(* IEC 61131-3 sources: netflux/Codesys_V3/NETFLUX, 14 files *)

(* ---- DUT_INPUTS.st ---- *)
TYPE DUT_INPUTS :
STRUCT
	Conv1_fb_pulse : BIT; //Pulse position sensor
	conv2_fb_pulse : BIT; //Pulse position sensor
	SPARE_INPUT_01 : BIT; //Spare bit
	SPARE_INPUT_02 : BIT; //Spare bit
	SPARE_INPUT_03 : BIT; //Spare bit
	SPARE_INPUT_04 : BIT; //Spare bit
	SPARE_INPUT_05 : BIT; //Spare bit
	SPARE_INPUT_06 : BIT; //Spare bit
	PS1_fb : BIT; //Sensor feedback signal
	PS2_fb : BIT; //Sensor feedback signal
	SPARE_INPUT_07 : BIT; //Spare bit
	SPARE_INPUT_08 : BIT; //Spare bit
	SPARE_INPUT_09 : BIT; //Spare bit
	SPARE_INPUT_10 : BIT; //Spare bit
	SPARE_INPUT_11 : BIT; //Spare bit
	SPARE_INPUT_12 : BIT; //Spare bit
	RDS1_fb_rised : BIT; //Rising divert at raised position
	RDS1_fb_initial : BIT; //Rising divert at initial position
	SPARE_INPUT_13 : BIT; //Spare bit
	SPARE_INPUT_14 : BIT; //Spare bit
	SPARE_INPUT_15 : BIT; //Spare bit
	SPARE_INPUT_16 : BIT; //Spare bit
	SPARE_INPUT_17 : BIT; //Spare bit
	SPARE_INPUT_18 : BIT; //Spare bit
	SPARE_INPUT_19 : BIT; //Spare bit
	SPARE_INPUT_20 : BIT; //Spare bit
	SPARE_INPUT_21 : BIT; //Spare bit
	SPARE_INPUT_22 : BIT; //Spare bit
	SPARE_INPUT_23 : BIT; //Spare bit
	SPARE_INPUT_24 : BIT; //Spare bit
	SPARE_INPUT_25 : BIT; //Spare bit
	SPARE_INPUT_26 : BIT; //Spare bit
	SPARE_INPUT_27 : BIT; //Spare bit
	SPARE_INPUT_28 : BIT; //Spare bit
	SPARE_INPUT_29 : BIT; //Spare bit
	SPARE_INPUT_30 : BIT; //Spare bit

END_STRUCT
END_TYPE

(* ---- DUT_OUTPUTS.st ---- *)
TYPE DUT_OUTPUTS :
STRUCT
	Conv1_cmd_fwd : BIT; //Run conveyor forward
	conv2_cmd_fwd : BIT; //Run conveyor forward
	Conv1_cmd_bwd : BIT; //Run conveyor backward
	conv2_cmd_bwd : BIT; //Run conveyor backward
	SPARE_OUTPUT_01 : BIT; //Spare bit
	SPARE_OUTPUT_02 : BIT; //Spare bit
	SPARE_OUTPUT_03 : BIT; //Spare bit
	SPARE_OUTPUT_04 : BIT; //Spare bit
	em1_cmd_emit : BIT; //Trigger item spawn
	destroyer_cmd_on : BIT; //Enable destroyer
	SPARE_OUTPUT_05 : BIT; //Spare bit
	SPARE_OUTPUT_06 : BIT; //Spare bit
	SPARE_OUTPUT_07 : BIT; //Spare bit
	SPARE_OUTPUT_08 : BIT; //Spare bit
	SPARE_OUTPUT_09 : BIT; //Spare bit
	SPARE_OUTPUT_10 : BIT; //Spare bit
	RDS1_cmd_left : BIT; //Command divert left (belt forward)
	RDS1_cmd_right : BIT; //Command divert right (belt backward)
	SPARE_OUTPUT_11 : BIT; //Spare bit
	SPARE_OUTPUT_12 : BIT; //Spare bit
	SPARE_OUTPUT_13 : BIT; //Spare bit
	SPARE_OUTPUT_14 : BIT; //Spare bit
	SPARE_OUTPUT_15 : BIT; //Spare bit
	SPARE_OUTPUT_16 : BIT; //Spare bit
	SPARE_OUTPUT_17 : BIT; //Spare bit
	SPARE_OUTPUT_18 : BIT; //Spare bit
	SPARE_OUTPUT_19 : BIT; //Spare bit
	SPARE_OUTPUT_20 : BIT; //Spare bit
	SPARE_OUTPUT_21 : BIT; //Spare bit
	SPARE_OUTPUT_22 : BIT; //Spare bit
	SPARE_OUTPUT_23 : BIT; //Spare bit
	SPARE_OUTPUT_24 : BIT; //Spare bit
	SPARE_OUTPUT_25 : BIT; //Spare bit
	SPARE_OUTPUT_26 : BIT; //Spare bit

END_STRUCT
END_TYPE

(* ---- DUT_RECV_DATA.st ---- *)
{attribute 'pack_mode' := '0'}
TYPE DUT_RECV_DATA :
STRUCT
		byteArray :	ARRAY[0..50] OF BYTE;
		some_INT :	INT;
		some_TIME :	TIME;
		some_REAL :	REAL;
		b1 :	BYTE ;
		b2 :	BYTE ;
		b3 :	BYTE ;

END_STRUCT
END_TYPE

(* ---- ENUM_NetfluxSocketState.st ---- *)
TYPE ENUM_NetfluxSocketState :
(
    IDLE := 0,
    CREATE := 10,
    BIND := 20,
    NONBLOCK := 30,
    RUNNING := 40,
    ERROR := 99
) INT;
END_TYPE

(* ---- GVL.st ---- *)
{attribute 'qualified_only'}
VAR_GLOBAL
	data_send :  DUT_OUTPUTS;
	data_recv :  DUT_INPUTS;
END_VAR

(* ---- fbNetflux_Recieve.st ---- *)
(*
    Function Block: fbPUDP_Recieve
    Description: Manages the receiving part of a UDP communication.
                 It uses a sequence number to discard duplicate or out-of-order packets
                 and a watchdog timer to detect communication loss. It provides outputs
                 needed by a corresponding Send block.
*)
FUNCTION_BLOCK fbNetflux_Recieve
VAR_INPUT
    // --- Connection Parameters ---
    i_uiLocalPort : UINT;   // Local UDP port to listen on.

    // --- Data Reception Parameters ---
	i_ptrReceiveData : POINTER TO BYTE; // Pointer to the destination buffer where the received data payload will be stored.
	i_uiSizeReceiveData : UINT;         // The exact size of the data payload to copy. The user is responsible for ensuring this size matches the sender's payload.

    // --- Watchdog Parameters ---
    i_tWatchInterval : TIME := T#1S;    // Watchdog timeout. If no new valid packet arrives within this interval, o_bError is set.
    i_xKeepValuesOnTimeout : BOOL;      // If TRUE, the last received values are kept in the destination buffer on watchdog timeout. If FALSE, the buffer is cleared for safety.
END_VAR
VAR_OUTPUT
    o_xError: BOOL;        // Becomes TRUE if no valid packet has been received, if the watchdog has timed out, or if a library error occurs.
    o_eErrorID: NBS.ERROR; // Propagates the specific error code from the underlying NBS library if an error occurs.
	o_hPeer: LWORD;         // Outputs the handle of the UDP peer. This is required by the corresponding Send block to use the same socket.
	o_bPartnerSeqNumber : BYTE; // Outputs the last received sequence number from the partner. This is needed by the Send block to send it back as a feedback sequence number.
	o_bCurrentFeedbackSeqNumber : BYTE; // Stores the feedback sequence number from the current valid packet. Used by the watchdog.
END_VAR
VAR
	// --- Internal state flags ---
	s_xFirstPacketReceived : BOOL;      // Flag to track if at least one valid packet has been received since startup or last timeout.
    s_xWatchdogTimeout : BOOL;          // Flag set by the watchdog timer when no new packet arrives in time.

    // --- UDP library instances ---
    s_fbPeer: NBS.UDP_Peer := (xEnable := TRUE); // Manages the UDP socket itself.
	s_fbUDPReceive : NBS.UDP_Receive;            // Handles the continuous reception of data into the internal buffer.
    s_tonWatchdog : TON;                         // Watchdog timer to detect communication loss.

    // --- Internal receive buffer ---
    s_aRecvBuffer: ARRAY[0..1460] OF BYTE;       // Raw buffer that receives the entire UDP packet.
	s_ptrRecvBuffer : POINTER TO BYTE := ADR(s_aRecvBuffer);
	s_szRecvBuffer : UINT := SIZEOF(s_aRecvBuffer);

	// --- Sequence number handling ---
	s_bPreviousRecvSeqNumber : BYTE;    // Stores the sequence number of the last processed packet to detect new ones.

    s_bPreviousFeedbackSeqNumber : BYTE;// Stores the feedback sequence number from the previous cycle to detect changes.
END_VAR
VAR_TEMP
    xIsNewPacket : BOOL;                // Temporary flag to indicate if a received packet is newer than the last processed one.
END_VAR

// === IMPLEMENTATION ===
(*
    This function block receives data via UDP and writes it into a specified destination buffer.

    Expected UDP Payload Structure:
    - Byte 0: Sequence Number (rolls over from 255 to 0). Used to identify new/unique packets.
    - Byte 1: Feedback Sequence Number. A copy of the sender's own receive sequence number. Used here for the watchdog.
    - Byte 2...N: The actual data payload.

    How it works:
    1. It continuously listens for incoming UDP packets on the specified port using the NBS library blocks.
    2. It checks for a new packet by comparing the sequence number (Byte 0) of the incoming packet with the last one processed.
    3. A robust sequence number validation handles counter wrap-around and rejects old, duplicate, or out-of-order packets.
    4. For valid new packets, a fixed-size data payload (defined by 'i_uiSizeReceiveData') is copied from the internal buffer to the user-provided destination buffer.
    5. A watchdog timer monitors the reception of valid packets. If no new packet arrives within 'i_tWatchInterval', an error is flagged.
    6. If the watchdog expires, the behavior is controlled by 'i_bKeepValuesOnTimeout' (either clear the destination buffer or keep the last valid data).
*)

// 1. Initialize and open the UDP Peer on the specified local port.
s_fbPeer(uiPort:=i_uiLocalPort);
// 1a. Output the peer handle so a corresponding Send block can use the same socket.
o_hPeer := s_fbPeer.hPeer;

// 2. Execute the UDP_Receive instruction to listen for data. This block continuously updates s_aRecvBuffer with the latest received packet.
s_fbUDPReceive(
	xEnable:= s_fbPeer.xActive,
	hPeer:= s_fbPeer.hPeer,
	szSize:= s_szRecvBuffer,
	pData:= s_ptrRecvBuffer);

// 3. Check for a new packet by detecting a change in the sequence number byte.
IF s_aRecvBuffer[0] <> s_bPreviousRecvSeqNumber THEN
	// 3a. Pass the received sequence number to the output immediately. The Send block will use this for feedback.
	o_bPartnerSeqNumber := s_aRecvBuffer[0];

    // A packet with a different sequence number has arrived.
    // Now, validate if it's logically NEWER than the last one, handling the 8-bit counter wrap-around.
    // This prevents processing old packets that may arrive out of order.
    // A packet is considered "new" if it's the first one, its number is slightly ahead, or it has wrapped around.
    xIsNewPacket := NOT s_xFirstPacketReceived OR
        (s_aRecvBuffer[0] > s_bPreviousRecvSeqNumber AND s_aRecvBuffer[0] - s_bPreviousRecvSeqNumber < 128) OR
        (s_aRecvBuffer[0] < s_bPreviousRecvSeqNumber AND s_bPreviousRecvSeqNumber - s_bPreviousRecvSeqNumber > 128);

	IF xIsNewPacket THEN
        // --- Process Valid New Packet ---
        s_xFirstPacketReceived := TRUE;
        o_bCurrentFeedbackSeqNumber := s_aRecvBuffer[1]; // Store feedback number for the watchdog.

        // Copy the data payload (starting from the 3rd byte) from the internal buffer to the destination buffer.
        MEMUtils.MemCpy(pbyDest:= i_ptrReceiveData,
                        pbySrc:= ADR(s_aRecvBuffer[2]),
                        dwSize:= i_uiSizeReceiveData);

        // IMPORTANT: Update the previous sequence number *only after* successfully processing a valid new packet.
        s_bPreviousRecvSeqNumber := s_aRecvBuffer[0];
	END_IF;
END_IF;

// 4. Watchdog timer logic. The timer is active if a valid packet has been received but no new one has arrived.
// It checks if the feedback sequence number has changed. A change indicates the partner has received our data, implying the connection is alive.
s_tonWatchdog(
    IN:= (o_bCurrentFeedbackSeqNumber = s_bPreviousFeedbackSeqNumber) AND s_xFirstPacketReceived,
    PT:= i_tWatchInterval,
    Q=> s_xWatchdogTimeout);

// Update the previous feedback number for the next cycle's comparison.
s_bPreviousFeedbackSeqNumber := o_bCurrentFeedbackSeqNumber;

// 5. Handle watchdog timeout.
IF s_xWatchdogTimeout AND NOT i_xKeepValuesOnTimeout THEN
    // If the timeout occurs and we are not keeping values, clear the destination buffer for safety.
    MEMUtils.MemSet(pbyBuffer:= i_ptrReceiveData,
                    byValue:= 0,
                    dwSize:= i_uiSizeReceiveData);

    // Reset the state to require a new "first" packet.
    s_xFirstPacketReceived := FALSE;
END_IF;

// 6. Aggregate final error output. An error exists if we haven't received a valid packet yet, the watchdog timed out, or a library block has an error.
o_xError := NOT s_xFirstPacketReceived OR s_xWatchdogTimeout OR s_fbPeer.xError OR s_fbUDPReceive.xError;

// 7. Propagate specific error codes from the underlying library for easier debugging.
IF s_fbPeer.xError THEN
    o_eErrorID := s_fbPeer.eError;
ELSIF s_fbUDPReceive.xError THEN
    o_eErrorID := s_fbUDPReceive.eError;
END_IF;

(* ---- fbNetflux_Send.st ---- *)
(*
    Function Block: fbPUDP_Send
    Description: Manages the sending part of a UDP communication.
                 It periodically sends a packet containing a sequence number, a feedback
                 sequence number, and the data payload. It is designed to work in tandem
                 with the fbPUDP_Recieve block.
*)
FUNCTION_BLOCK fbNetflux_Send
VAR_INPUT
    // --- Connection Parameters ---
	i_uiRemotePort : UINT;      // The UDP port of the remote partner.
	i_sIPaddress : STRING[15];  // The IP address of the remote partner.
	i_tSendInterval : TIME := T#5MS; // The interval at which to send packets.

    // --- Link to Recieve Block ---
	i_hPeer: LWORD;              // The handle of the UDP peer, obtained from the fbPUDP_Recieve block.
	i_bPartnerSeqNumber : BYTE; // The last sequence number received from the partner, provided by fbPUDP_Recieve. This is sent back for feedback.

    // --- Data to Send ---
	i_ptrSendData : POINTER TO BYTE; // Pointer to the source buffer containing the data payload to send.
	i_uiSizeSendData : UINT;         // The size of the data payload to send.
END_VAR
VAR_OUTPUT
	o_bSequenceNumber : BYTE;   // The internal sequence number for outgoing packets. Increments with each send.
    o_bError: BOOL;        // Becomes TRUE if a library error occurs during sending.
    o_eErrorID: NBS.ERROR; // Propagates the specific error code from the underlying NBS library if an error occurs.
END_VAR
VAR
    // --- UDP library instances ---
	s_fbUDPSend : NBS.UDP_Send;
	s_tonSendPeriod : TON;      // Timer to trigger sending at the specified interval.
	s_IPaddress : NBS.IP_ADDR;  // Structure to hold the remote IP address.

    // --- Internal state ---
	s_xSend : BOOL;             // Trigger flag for sending, controlled by the timer.
	s_xInit : BOOL := TRUE;     // Flag for one-time initialization on the first scan.

	// --- Internal send buffer ---
    s_aSendBuffer: ARRAY[0..1460] OF BYTE; // Raw buffer used to construct the entire UDP packet before sending.
	s_ptrSendBuffer : POINTER TO BYTE := ADR(s_aSendBuffer);
	s_szTotalPacketSize : UINT; // Holds the total size of the packet to be sent (Header + Payload).
END_VAR

// === IMPLEMENTATION ===
(*
    This function block sends data via UDP.

    UDP Payload Structure created by this block:
    - Byte 0: s_bSequenceNumber (This block's own incrementing sequence number).
    - Byte 1: i_bPartnerSeqNumber (The sequence number received from the partner, used as feedback).
    - Byte 2...N: The actual data payload from i_ptrSendData.

    How it works:
    1. On the first scan, it initializes the remote IP address and calculates the total packet size. This is an optimization to avoid repeated calculations.
    2. A timer triggers the sending process at the interval specified by 'i_tSendInterval'.
    3. When triggered, it constructs the packet header in an internal buffer (s_aSendBuffer) and copies the user data payload.
    4. It increments its own sequence number for each packet.
    5. It calls the NBS.UDP_Send function block to transmit the constructed packet.
    6. It monitors for errors from the library and exposes them through the outputs.
*)

// 1. One-time initialization on the first scan.
IF s_xInit THEN
	// Set the remote IP address and calculate the total packet size.
    // This is done only once for efficiency.
	s_IPaddress.sAddr := i_sIPaddress;
    s_szTotalPacketSize := i_uiSizeSendData + 2; // Payload size + 2 bytes for the header.

	s_xInit := FALSE;
END_IF;

// 2. Generate a periodic trigger for sending. s_xSend will be TRUE for one cycle every i_tSendInterval.
s_tonSendPeriod(IN:= NOT s_xSend, PT:= i_tSendInterval, Q=> s_xSend);

// 3. When the timer triggers, prepare the packet.
IF s_xSend THEN
    // --- Construct the packet header ---
    o_bSequenceNumber := o_bSequenceNumber + 1; // Increment our own sequence number.
    s_aSendBuffer[0] := o_bSequenceNumber;      // Byte 0: Our sequence number.
    s_aSendBuffer[1] := i_bPartnerSeqNumber;    // Byte 1: The partner's sequence number (feedback).

    // --- Copy the data payload into the buffer after the header ---
    MEMUtils.MemCpy(pbyDest:= ADR(s_aSendBuffer[2]),
                    pbySrc:= i_ptrSendData,
                    dwSize:= i_uiSizeSendData);
END_IF;

// 4. Execute the UDP_Send instruction.
// It is called continuously, but the xExecute flag ensures it only acts when triggered.
s_fbUDPSend(
	xExecute:= s_xSend,
	udiTimeOut:= 50000, // Timeout in microseconds (50ms)
	hPeer:= i_hPeer,
	ipAddr:= s_IPaddress,
	uiPort:= i_uiRemotePort,
	szSize:= s_szTotalPacketSize,
	pData:= s_ptrSendBuffer);

// 5. Handle error outputs from the library block.
o_bError := s_fbUDPSend.xError;
IF o_bError THEN
    o_eErrorID := s_fbUDPSend.eError;
END_IF;

(* ---- fbNetflux_Socket.st ---- *)
(*
    Function Block: fbNetflux_Socket (v5 - Final Mixed Signatures)
    Description: Unified UDP Sender/Receiver using SysSocket logic.
                 Signatures Tuned:
                 - RecvFrom/SendTo/InetAddr: REQUIRE pResult.
                 - Bind/Ioctl: NO pResult (3 args).
 *)
FUNCTION_BLOCK fbNetflux_Socket
VAR_INPUT
    xEnable: BOOL := TRUE;
    xReconnect: BOOL := FALSE;  // Rising edge triggers reconnection

    // --- Network Config ---
    sRemoteIP: STRING(15);
    uiRemotePort: UINT;
    uiLocalPort: UINT;
    tSendInterval: TIME := T#2MS;

    // --- Data Handlers ---
    ptrSendData: POINTER TO BYTE;
    uiSizeSendData: UDINT;

    ptrRecvData: POINTER TO BYTE;
    uiSizeRecvData: UDINT;
END_VAR
VAR_OUTPUT
    xError: BOOL;
    xConnected: BOOL;

    uiPacketsReceivedPerCycle: UINT;
    tRoundTripTime: TIME;
    bLastPartnerSeq: BYTE;

    // Statistics
    udiTxCount: UDINT;
    udiRxCount: UDINT;

    // Statistics - Optional (calculated when Statistics() is called)
    tPartnerTxPeriod: TIME;      // Partner's transmission period
    tOwnRealTxPeriod: TIME;      // Own real transmission period
    tInstantRTT: TIME;           // Instantaneous RTT
    uiInstantRxSkipped: UINT;    // Instantaneous RX skipped packets

    // Diagnostics
    eCurrentState: ENUM_NetfluxSocketState;  // Current state for debugging
END_VAR
VAR
    hSocket: UDINT := 16#FFFFFFFF;

    saLocal: SOCKADDRESS;
    saRemote: SOCKADDRESS;

    eState: ENUM_NetfluxSocketState := ENUM_NetfluxSocketState.IDLE;

    xFirstCycle: BOOL := TRUE;  // Flag to detect cold start / program reload
    udiInitCounter: UDINT := 0;  // Counter for reliable cold start detection

    tonSend: TON;
    tonWatchdog: TON := (PT := T#1s);

    aRecvBuf: ARRAY[0..1500] OF BYTE;
    aSendBuf: ARRAY[0..1500] OF BYTE;

    bOwnSeq: BYTE;
    bLastRecvSeq: BYTE;

    // --- Helpers ---
    diRes: DINT;
    diRecvBytes: DINT;
    diSentBytes: DINT;
    diDummy: DINT;
    xi: DINT;

    xNewData: BOOL;

    nrResult: DINT;

    // --- Statistics Internal Variables ---
    tLastRxTime: TIME;           // Timestamp of last received packet
    tLastTxTime: TIME;           // Timestamp of last sent packet
    bPrevRecvSeq: BYTE;          // Previous received sequence number
    bPrevOwnSeq: BYTE;           // Previous own sequence number
    xFirstRx: BOOL := TRUE;      // Flag for first reception
    xFirstTx: BOOL := TRUE;      // Flag for first transmission

    // --- Reconnect Edge Detection ---
    xReconnect_prev: BOOL := FALSE;  // Previous state of xReconnect

    // --- Error Recovery ---
    tonErrorRecovery: TON := (PT := T#5s);  // Auto-recovery timer for ERROR state
END_VAR

// === IMPLEMENTATION ===
// Cold Start Detection: Force reset on program reload
// Use both flag and counter for reliability (CODESYS may not reset BOOL := TRUE on download)
IF xFirstCycle OR udiInitCounter = 0 THEN
    xFirstCycle := FALSE;
    udiInitCounter := 1;

    // Check if socket handle exists and might be stale
    IF hSocket <> 16#FFFFFFFF THEN
        xi := 0;
        diDummy := SIZEOF(xi);
		{warning disable C0196}
        diRes := SysSockGetOption(hSocket, SOCKET_SOL, SOCKET_SO_TYPE, ADR(xi), ADR(diDummy));

        // If GetOption fails, socket is invalid/stale
        IF diRes <> 0 THEN
            // Socket is stale, just reset handle
            hSocket := 16#FFFFFFFF;
        ELSE
            // Socket seems valid but we're restarting - close it properly
            THIS^.CloseSocket();
        END_IF
    END_IF

    // Force clean restart
    eState := ENUM_NetfluxSocketState.IDLE;
    xError := FALSE;
    xConnected := FALSE;
END_IF

// Manual Reconnect Trigger: Detect rising edge on xReconnect
IF xReconnect AND NOT xReconnect_prev THEN
    // Close existing socket
    THIS^.CloseSocket();

    // Reset to IDLE to trigger reconnection
    eState := ENUM_NetfluxSocketState.IDLE;
    xError := FALSE;
    xConnected := FALSE;
END_IF
xReconnect_prev := xReconnect;

CASE eState OF
    ENUM_NetfluxSocketState.IDLE: // Idle / Init
        IF xEnable THEN
            eState := ENUM_NetfluxSocketState.CREATE;
        END_IF

    ENUM_NetfluxSocketState.CREATE: // Create Socket
        hSocket := SysSockCreate(SOCKET_AF_INET, SOCKET_DGRAM, SOCKET_IPPROTO_UDP, ADR(nrResult));

        IF hSocket <> 16#FFFFFFFF THEN
            // Set SO_REUSEADDR to allow port reuse (critical for reconnection!)
            // This allows binding to a port in TIME_WAIT state
            xi := 1;
            diRes := SysSockSetOption(hSocket, SOCKET_SOL, SOCKET_SO_REUSEADDR, ADR(xi), SIZEOF(xi));

            // Try to set SO_REUSEPORT as well (may not be available on all systems)
            // This allows multiple sockets to bind to the same port
            // Ignore errors as this is optional
            IF diRes = 0 THEN
                xi := 1;
                diDummy := SysSockSetOption(hSocket, SOCKET_SOL, 15 (*SO_REUSEPORT*), ADR(xi), SIZEOF(xi));
                // Continue even if SO_REUSEPORT fails
            END_IF

            IF diRes = 0 THEN
                eState := ENUM_NetfluxSocketState.BIND;
            ELSE
                // Failed to set socket option, close and error
                THIS^.CloseSocket();
                eState := ENUM_NetfluxSocketState.ERROR;
            END_IF
        ELSE
            eState := ENUM_NetfluxSocketState.ERROR;
        END_IF

    ENUM_NetfluxSocketState.BIND: // Bind TO:
        saLocal.sin_family := SOCKET_AF_INET;
        saLocal.sin_port := SysSockHtons(uiLocalPort);
        saLocal.sin_addr.ulAddr := SOCKET_INADDR_ANY;

        // SysSockBind: 3 args (Handle, pAddr, iSize) - NO pResult
        diRes := SysSockBind(hSocket, ADR(saLocal), SIZEOF(saLocal));

        IF diRes = 0 THEN
            eState := ENUM_NetfluxSocketState.NONBLOCK;
        ELSE
            eState := ENUM_NetfluxSocketState.ERROR;
        END_IF

    ENUM_NetfluxSocketState.NONBLOCK: // Non-Blocking
        xi := 1;
        // SysSockIoctl: 3 args (Handle, Cmd, pArg) - NO pResult
        diRes := SysSockIoctl(hSocket, SOCKET_FIONBIO, ADR(xi));

        IF diRes = 0 THEN
            eState := ENUM_NetfluxSocketState.RUNNING;

            saRemote.sin_family := SOCKET_AF_INET;
            saRemote.sin_port := SysSockHtons(uiRemotePort);
            // InetAddr: 2 args (String, pResult) - WITH pResult
            saRemote.sin_addr.ulAddr := SysSockInetAddr(sRemoteIP, ADR(nrResult));
        ELSE
            eState := ENUM_NetfluxSocketState.ERROR;
        END_IF

    ENUM_NetfluxSocketState.RUNNING: // RUNNING
        xConnected := NOT tonWatchdog.Q;
        IF NOT xEnable THEN
            THIS^.CloseSocket();
            eState := ENUM_NetfluxSocketState.IDLE;
            RETURN;
        END_IF

        // RECV LOOP
        uiPacketsReceivedPerCycle := 0;

        FOR xi := 0 TO 20 DO
            // RecvFrom: 7 args (Handle, Buf, Size, Flags, Addr, Size, pResult)
            diRecvBytes := SysSockRecvFrom(hSocket, ADR(aRecvBuf), SIZEOF(aRecvBuf), 0, ADR(saRemote), SIZEOF(saRemote), ADR(nrResult));

            IF diRecvBytes > 0 THEN
                uiPacketsReceivedPerCycle := uiPacketsReceivedPerCycle + 1;
                udiRxCount := udiRxCount + 1; // Update Stats

                IF diRecvBytes >= 2 THEN
                    bLastRecvSeq := aRecvBuf[0];
                    bLastPartnerSeq := bLastRecvSeq;

                    // Capture timestamp for statistics
                    tLastRxTime := TIME();

                    tonWatchdog(IN := FALSE);

                    IF ptrRecvData <> 0 AND uiSizeRecvData > 0 THEN
                         IF UDINT_TO_INT(uiSizeRecvData) <= (diRecvBytes - 2) THEN
                            SysMemCpy(ptrRecvData, ADR(aRecvBuf[2]), uiSizeRecvData);
                         END_IF
                    END_IF
                END_IF
            ELSE
                EXIT;
            END_IF
        END_FOR

        tonWatchdog(IN := TRUE);

        // Execute Statistics
        THIS^.Statistics();

    ENUM_NetfluxSocketState.ERROR: // Error
        xError := TRUE;

        // Auto-recovery: Try to reconnect after timeout if still enabled
        tonErrorRecovery(IN := xEnable);

        IF tonErrorRecovery.Q THEN
            // Close socket if it exists
            THIS^.CloseSocket();

            // Reset to IDLE to retry connection
            eState := ENUM_NetfluxSocketState.IDLE;
            xError := FALSE;
            tonErrorRecovery(IN := FALSE);  // Reset timer
        END_IF

        // If disabled, reset error state
        IF NOT xEnable THEN
            tonErrorRecovery(IN := FALSE);
            eState := ENUM_NetfluxSocketState.IDLE;
            xError := FALSE;
        END_IF

END_CASE

// Update diagnostic output
eCurrentState := eState;

(* ---- fbNetflux_Statistics.st ---- *)
(*
    Function Block: fbPUDP_Statistics_V2
    Description: Calculates communication statistics with alternative logic.
                 - Intervals are measured by timing the duration of a full sequence number cycle (0-255).
                 - RTT is measured by tracking a single sequence number until its acknowledgment is received.
                 - Packet loss is calculated by detecting gaps in sequence numbers.
*)
FUNCTION_BLOCK fbNetflux_Statistics
VAR_INPUT
	i_xStatReset : BOOL; // Resets all statistical data.
	i_bRecvSeqNumber : BYTE; // The sequence number from the partner's last received packet.
	i_bSequenceNumber : BYTE;   // Your own send sequence number from the Send block.
	i_bFeedbackSeqNumber : BYTE; // The feedback from the partner (your own sequence number being returned).
    i_rTaskCycle : REAL; // Standard precision cycle time in ms
END_VAR
VAR_OUTPUT
    // --- Interval Statistics (calculated over a full ~256-packet cycle) ---
    o_rAvgPartnerInterval : REAL;       // Average time between packets received from the partner.
    o_rAvgOwnInterval : REAL;           // Average time between packets sent by this PLC.

    // --- Round Trip Time (RTT) Statistics ---
    o_rLastRTT : REAL;                  // The last measured round trip time.

    // --- Packet Loss Statistics ---
    o_bTotalPartnerLostPackets : BYTE;     // Total packets lost from the partner (gaps in i_bPartnerSeqNumber).
    o_bTotalFeedbackLostPackets : BYTE;     // Total acknowledgments lost from the partner (gaps in i_bCurrentFeedbackSeqNumber).
END_VAR
VAR
    // --- Triggers ---
    s_trigReset : R_TRIG;
    s_trigNewRecvPacket : R_TRIG;
    s_trigNewSendPacket : R_TRIG;
    s_trigFeedbackSeqNumber : R_TRIG;
	s_trigSendPacketRound : R_TRIG;
	s_trigRecvPacketRound : R_TRIG;
	s_trigFeedbackPacketRound : R_TRIG;

    // --- Own Send Interval Internals ---
    s_rOwnCycleCounter : REAL;
    s_bPrevSendSeqNumber : BYTE;
    s_xOwnCycleTiming : BOOL;

    // --- Partner Interval Internals ---
    s_rPartnerCycleCounter : REAL;
    s_bPrevRecvSeqNumber : BYTE;

    // --- Packet Loss Feedback Internals ---
    s_bPrevFeedBackSeqNumber : BYTE;
    s_xFirstPartnerPacket : BOOL := TRUE;
    s_xFirstAckPacket : BOOL := TRUE;

	// --- RTT Internals ---
    s_rRTTCounter : REAL;
    s_bRTT_TrackedSeqNum : BYTE;
END_VAR
VAR_TEMP
    uiLostCount : UINT;
END_VAR

// === IMPLEMENTATION ===
//Triggers
s_trigReset(CLK:= i_xStatReset);
s_trigNewRecvPacket(CLK:= i_bRecvSeqNumber <> s_bPrevRecvSeqNumber);
s_trigNewSendPacket(CLK:= i_bSequenceNumber <> s_bPrevSendSeqNumber);
s_trigFeedbackSeqNumber(CLK:= i_bFeedBackSeqNumber <> s_bPrevFeedBackSeqNumber);
s_trigSendPacketRound(CLK:= i_bSequenceNumber >= 0 AND i_bSequenceNumber < 3);
s_trigRecvPacketRound(CLK:= i_bRecvSeqNumber >= 0 AND i_bRecvSeqNumber < 5);
s_trigFeedbackPacketRound(CLK:= i_bFeedbackSeqNumber >= 0 AND i_bFeedbackSeqNumber < 15);

//Average time between packets received from the partner
IF s_trigSendPacketRound.Q THEN
	o_rAvgOwnInterval := s_rOwnCycleCounter / 256.0 - 2.0 * i_rTaskCycle;
	s_rOwnCycleCounter := 0.0;
ELSE
	s_rOwnCycleCounter := s_rOwnCycleCounter + i_rTaskCycle;
END_IF
//Average time between packets sent by this PLC.
IF s_trigRecvPacketRound.Q THEN
	o_rAvgPartnerInterval := s_rPartnerCycleCounter / 256.0 - 2.0 * i_rTaskCycle;
	s_rPartnerCycleCounter := 0.0;
ELSE
	s_rPartnerCycleCounter := s_rPartnerCycleCounter + i_rTaskCycle;
END_IF

// Total packets lost from the feedback (gaps in i_bFeedBackSeqNumber).
IF i_bFeedBackSeqNumber - s_bPrevFeedBackSeqNumber > 1 THEN
	o_bTotalFeedbackLostPackets := o_bTotalFeedbackLostPackets + (i_bFeedBackSeqNumber - s_bPrevFeedBackSeqNumber - 1);
END_IF

IF s_trigFeedbackPacketRound.Q THEN
	o_bTotalFeedbackLostPackets := 0;
END_IF

// Total packets lost from the partner
IF i_bRecvSeqNumber - s_bPrevRecvSeqNumber > 1 THEN
	o_bTotalPartnerLostPackets := o_bTotalPartnerLostPackets + (i_bRecvSeqNumber - s_bPrevRecvSeqNumber - 1);
END_IF

IF s_trigRecvPacketRound.Q THEN
	o_bTotalPartnerLostPackets := 0;
END_IF

// The last measured round trip time.
IF s_trigNewSendPacket.Q AND s_bRTT_TrackedSeqNum = 0 THEN
	s_bRTT_TrackedSeqNum := i_bSequenceNumber;
	s_rRTTCounter := 0.0;
ELSE
	s_rRTTCounter := s_rRTTCounter + i_rTaskCycle;
END_IF

IF s_bRTT_TrackedSeqNum = i_bFeedbackSeqNumber THEN
	o_rLastRTT := s_rRTTCounter;
	s_bRTT_TrackedSeqNum := 0;
END_IF

//Auxilary save previous values
s_bPrevRecvSeqNumber := i_bRecvSeqNumber;
s_bPrevSendSeqNumber := i_bSequenceNumber;
s_bPrevFeedBackSeqNumber := i_bFeedBackSeqNumber;

(* ---- fbTaskInfo.st ---- *)
(*
Function Block: fbTaskInfo
Purpose: Retrieves and processes current task timing information. Works only with TaskCyclic.
Outputs:
  - lrTaskCycle: Task cycle time in milliseconds (LREAL)
  - rTaskCycle: Task cycle time in milliseconds (REAL)
  - xTaskCycle: Task cycle time as TIME value. works only with task >= 1ms
*)
FUNCTION_BLOCK fbTaskInfo
VAR
    _stTaskInfo : POINTER TO Task_Info2;              // Pointer to task information structure
    _IecTaskGetCurrent : UDINT;                      // Result of IecTaskGetCurrent call
    _IecTaskGetInfo3 : UDINT;                        // Result of IecTaskGetInfo3 call
    _ptrIecTaskGetCurrent : POINTER TO UDINT := ADR(_IecTaskGetCurrent);    // Pointer for current task result
    _ptrIecTaskGetInfo3 : POINTER TO UDINT := ADR(_IecTaskGetInfo3);        // Pointer for task info result
END_VAR
VAR_OUTPUT
    lrTaskCycle : LREAL;       // High precision cycle time in ms
    rTaskCycle : REAL;         // Standard precision cycle time in ms
    tTaskCycle : TIME;         // Cycle time as TIME data type
END_VAR

// === IMPLEMENTATION ===
// Retrieve current task handle and task information
_stTaskInfo := IecTaskGetInfo3(
    hIecTask := IecTaskGetCurrent(pResult:= _ptrIecTaskGetCurrent),
    pResult:= _ptrIecTaskGetInfo3
);

// Process timing information based on task type
IF _stTaskInfo^.KindOfTask = 16#0 THEN        // Fixed interval execution, works only with TaskCyclic - KindOfTask
	 // Calculate cycle time including jitter for cyclic tasks
        lrTaskCycle := (DWORD_TO_LREAL(_stTaskInfo^.dwInterval) + DINT_TO_LREAL(_stTaskInfo^.iJitter)) / 1000.0;
        rTaskCycle := LREAL_TO_REAL(lrTaskCycle);
        tTaskCycle := REAL_TO_TIME(rTaskCycle);
END_IF

(* ---- fbNetflux_Socket.CloseSocket.st ---- *)
(*
    Method: CloseSocket
    Description: Properly closes the socket with shutdown to release port immediately
*)
METHOD PRIVATE CloseSocket
VAR
END_VAR

// === IMPLEMENTATION ===
// Shutdown socket first (releases port binding immediately)
IF hSocket <> 16#FFFFFFFF THEN
    // SOCKET_SD_BOTH = 2 (shutdown both send and receive)
    SysSockShutdown(hSocket, 2);

    // Now close the socket
    SysSockClose(hSocket);
    hSocket := 16#FFFFFFFF;
END_IF

(* ---- fbNetflux_Socket.send.st ---- *)
METHOD send : BOOL
VAR_INPUT
END_VAR
VAR
    nrResult: DINT; // Local result for SendTo
END_VAR

// === IMPLEMENTATION ===
tonSend(IN := NOT tonSend.Q, PT := tSendInterval);

IF tonSend.Q THEN
    bOwnSeq := bOwnSeq + 1;
    aSendBuf[0] := bOwnSeq;
    aSendBuf[1] := bLastRecvSeq;

    IF ptrSendData <> 0 AND uiSizeSendData > 0 THEN
         SysMemCpy(ADR(aSendBuf[2]), ptrSendData, uiSizeSendData);
    END_IF

    // SendTo: 7 args
	{warning disable C0196}
    SysSockSendTo(hSocket, ADR(aSendBuf), uiSizeSendData + 2, 0, ADR(saRemote), SIZEOF(saRemote), ADR(nrResult));

    // Update Stats
    udiTxCount := udiTxCount + 1;

    // Capture timestamp for statistics
    tLastTxTime := TIME();

    send := TRUE;
END_IF

(* ---- fbNetflux_Socket.Statistics.st ---- *)
METHOD Statistics: BOOL
VAR_INPUT
END_VAR
VAR
    tCurrentTime: TIME;
    tRxDelta: TIME;
    tTxDelta: TIME;
    iSeqDelta: INT;
END_VAR

// === IMPLEMENTATION ===
// This method calculates derived statistics based on timing and sequence information.
// It is optional and only calculates when called.

tCurrentTime := TIME();

// ========================================
// 1. Partner's Transmission Period
// ========================================
// Calculate time between received packets
IF NOT xFirstRx THEN
    tRxDelta := tCurrentTime - tLastRxTime;

    // Only update if we received a new packet (tRxDelta is reasonable)
    IF tRxDelta > T#0ms AND tRxDelta < T#10s THEN
        tPartnerTxPeriod := tRxDelta;
    END_IF
ELSE
    // First reception - no delta yet
    IF tLastRxTime > T#0ms THEN
        xFirstRx := FALSE;
    END_IF
END_IF

// ========================================
// 2. Own Real Transmission Period
// ========================================
// Calculate actual time between sent packets
IF NOT xFirstTx THEN
    tTxDelta := tCurrentTime - tLastTxTime;

    // Only update if we sent a new packet (tTxDelta is reasonable)
    IF tTxDelta > T#0ms AND tTxDelta < T#10s THEN
        tOwnRealTxPeriod := tTxDelta;
    END_IF
ELSE
    // First transmission - no delta yet
    IF tLastTxTime > T#0ms THEN
        xFirstTx := FALSE;
    END_IF
END_IF

// ========================================
// 3. Instantaneous RTT
// ========================================
// RTT is calculated based on the feedback sequence number
// The partner echoes our sequence in their packet (aSendBuf[1] = bLastRecvSeq)
// When we receive a packet, aRecvBuf[1] contains our sequence that partner echoed back
// RTT = time since we sent that sequence number

// For simplicity, we estimate RTT as half of the partner's transmission period
// This assumes symmetric delay and regular transmission
IF tPartnerTxPeriod > T#0ms THEN
    // Simple estimation: RTT ≈ Partner period / 2
    // More accurate would require tracking send times per sequence number
    tInstantRTT := tPartnerTxPeriod / 2;
END_IF

// Alternative RTT calculation based on sequence delta:
// If partner responds immediately, RTT ≈ our TX period
IF tOwnRealTxPeriod > T#0ms AND bLastRecvSeq <> 0 THEN
    // Use own period as RTT estimate if partner is responsive
    tInstantRTT := tOwnRealTxPeriod;
END_IF

// ========================================
// 4. Instantaneous RX Skipped Packets
// ========================================
// Calculate how many packets were skipped based on sequence number delta
IF bPrevRecvSeq <> 0 THEN
    // Calculate sequence delta (handle byte wraparound)
    iSeqDelta := BYTE_TO_INT(bLastRecvSeq) - BYTE_TO_INT(bPrevRecvSeq);

    // Handle wraparound: if delta is negative, add 256
    IF iSeqDelta < 0 THEN
        iSeqDelta := iSeqDelta + 256;
    END_IF

    // Skipped packets = delta - 1 (delta of 1 means consecutive, no skip)
    IF iSeqDelta > 1 THEN
        uiInstantRxSkipped := INT_TO_UINT(iSeqDelta - 1);
    ELSE
        uiInstantRxSkipped := 0;
    END_IF
ELSE
    uiInstantRxSkipped := 0;
END_IF

// Update previous sequence for next calculation
bPrevRecvSeq := bLastRecvSeq;

Statistics := TRUE;

(* ---- INLINE_CLOSE_ALTERNATIVE.st ---- *)
(*
    Alternative version without CloseSocket method
    Use this if method calls are not working
*)

// Replace THIS^.CloseSocket() with this inline code:

// Inline socket close
IF hSocket <> 16#FFFFFFFF THEN
    SysSockShutdown(hSocket, 2);  // SOCKET_SD_BOTH = 2
    SysSockClose(hSocket);
    hSocket := 16#FFFFFFFF;
END_IF
